SUBAPPLICATION AND_ZU (* Logisches UND (IN1 AND NOT IN2) für ZU-Bedingung *)
  (* Standard: 61499-2 *)
  (* Version 1.0, 2025-01-15, franz, Meisterschulen am Ostbahnhof *)
  PACKAGE MyLib::sys;
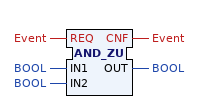
  EVENT_INPUT
    REQ;
  END_EVENT
  EVENT_OUTPUT
    CNF;
  END_EVENT
  VAR_INPUT
    IN1 : BOOL;
    IN2 : BOOL;
  END_VAR
  VAR_OUTPUT
    OUT : BOOL;
  END_VAR
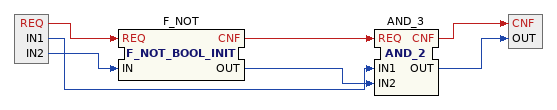
  FBS
    AND_3 : iec61131::bitwiseOperators::AND_2;
    F_NOT : iec61131::booleanOperators::F_NOT_BOOL_INIT;
  END_FBS
  EVENT_CONNECTIONS
    AND_3.CNF TO CNF;
    REQ TO F_NOT.REQ;
    F_NOT.CNF TO AND_3.REQ;
  END_CONNECTIONS
  DATA_CONNECTIONS
    IN1 TO AND_3.IN1;
    AND_3.OUT TO OUT;
    IN2 TO F_NOT.IN;
    F_NOT.OUT TO AND_3.IN2;
  END_CONNECTIONS
END_SUBAPPLICATION
